// TIA Portal V19 export
DATA_BLOCK "TIA_PN_FcP5020_DB"   // DB50153
// stored: InstanceOfName TIA_PN_FcP5020, InstanceOfType FB
"TIA_PN_FcP5020"
   // VAR_INPUT
   //    Enable : Bool;
   //    EnableDrive : Bool;
   //    ClearError : Bool;
   //    PressureCmd : Real;
   //    MaxSpeedLimit : Real;
   //    InputADDR : HW_IO;
   //    OutputADDR : HW_IO;
   // END_VAR
   // VAR_OUTPUT
   //    InOperation : Bool;
   //    MotorStarted : Bool;
   //    Error : Bool;
   //    Warning : Bool;
   //    DiagnosisCode : Word;
   //    Status : Word;
   //    PressureAct : Real;
   //    SpeedAct : Real;
   // END_VAR
   // VAR
   //    fbTON_TIME { S7_SetPoint := 'True'} : TON_TIME;
   //    bMbit0 : Bool;
   //    bMbit1 : Bool;
   //    bMbit2 : Bool;
   //    bMbit3 : Bool;
   //    bEnableRise : Bool;
   //    bErrorResetFall : Bool;
   //    bFBErrorFall : Bool;
   //    bClearErrorRise : Bool;
   //    stInputData { S7_SetPoint := 'True'} : "FCP_IN";
   //    stOutputData { S7_SetPoint := 'True'} : "FCP_OUT";
   //    hwInputADDR : HW_IO;
   //    hwOutputADDR : HW_IO;
   //    iStep : Int;
   //    iErrorStep : Int;
   //    iReturnVal : Int;
   //    wReturnVal : Word;
   //    bFBErrorPressureCmd : Bool;
   //    bFBErrorMaxSpeedLimit : Bool;
   //    bFBErrorDPRD_DPWR : Bool;
   //    bFcPError : Bool;
   //    bEFCError : Bool;
   //    bFcPWarning : Bool;
   //    bEFCWarning : Bool;
   //    rPressureCmdInternal : Real;
   //    rMaxSpeedLimtInternal : Real;
   //    bInternalRunTrigger : Bool;
   //    bInternalRun : Bool;
   // END_VAR
BEGIN
END_DATA_BLOCK
